TA08: A     #s_OS_UFO_Lost_Len_Change; // IF one-shot event UFO LNK lost due to length changed
      JCN   TA99;
      L     #s_Statistical.UFO_Lost_Length_Change; // THEN Increase number of times UFO LNK lost due to length changed
      L     1;
      +I    ;
      T     #s_Statistical.UFO_Lost_Length_Change;
TA99: NOP   0;
NETWORK
TITLE =UA: Deassign LNK in case of a deregister without HL reporting

      L     #t_ECS_Dereg_No_Rep_LNK;
      L     0;
      >I    ;
      JCN   UA01;

      CALL "FC_Deassign_LNK" (//Deassign the LNK
           i_LNK                    := #t_ECS_Dereg_No_Rep_LNK);

UA01: A(    ;
      L     #t_ECS_Dereg_No_Rep_LNK2;
      L     0;
      >I    ;
      )     ;
      A(    ;
      L     #t_ECS_Dereg_No_Rep_LNK;
      L     #t_ECS_Dereg_No_Rep_LNK2;
      <>I   ;
      )     ;
      JCN   UA99;

      CALL "FC_Deassign_LNK" (//Deassign the LNK
           i_LNK                    := #t_ECS_Dereg_No_Rep_LNK2);

UA99: NOP   0;
END_FUNCTION_BLOCK

